Staubli VAL3: acqSensorData.dtx

mdesc mNomSpeed
public CommParameter cSensorCommParm
  [0]
    num port
    string target
    num clients
    num endOfString
    num timeOut
    num baudRate
    string parity
    num bits
    num stopBits
    string mode
    string flowControl
    bool nagle
public sio sClientSensor
public num nSensitivity[6]
public num nZeroPoint[6]
public FlagStatus fSensorStatus
  [0]
    num ForceFlag
    num RosFlag
    num RobotFlag
